(* CODESYS project OOP example Advanced Array's.project

Project tree, tasks and I/O mapping:
  Device : CODESYS Control for Raspberry Pi SL, 3S - Smart Software Solutions GmbH, version 3.5.12.30
    application Application
      libraries: Standard, * (System); VisuDialogs, * (System); SysFile, 3.5.9.0 (System); AlarmManager, 3.5.12.0 (Intern)
      task MainTask (cyclic, interval 500 ms, priority 1, watchdog 1000 ms x 1) calls Arrays
      task VISU_TASK (cyclic, interval 100 ms, priority 31) calls VisuElems.Visu_Prg
      task AlarmManagerTask (cyclic, interval 250 ms, priority 31) calls AlarmManager.Alarm_Prg
      visualisation Arrays_Visu
      program Arrays [ST]
      Alarm Configuration
        alarm class Warning (priority 10, acknowledge REP)
        AlarmStorage
        text list AlarmGroup
        alarm group AlarmGroup
            7 [Warning]: Comparison NotEqual, ExpressionToCompare 0, Expression Arrays.arEngine[7].uiAlarm - "Engine 7 Alarm"
            4 [Warning]: Comparison NotEqual, ExpressionToCompare 0, Expression Arrays.arEngine[4].uiAlarm - "Engine 4 Alarm"
            5 [Warning]: Comparison NotEqual, ExpressionToCompare 0, Expression Arrays.arEngine[5].uiAlarm - "Engine 5 Alarm"
            2 [Warning]: Comparison NotEqual, ExpressionToCompare 0, Expression Arrays.arEngine[2].uiAlarm - "Engine 2 Alarm"
            3 [Warning]: Comparison NotEqual, ExpressionToCompare 0, Expression Arrays.arEngine[3].uiAlarm - "Engine 3 Alarm"
            0 [Warning]: Comparison NotEqual, ExpressionToCompare 0, Expression Arrays.arEngine[0].uiAlarm - "Engine 0 Alarm"
            1 [Warning]: Comparison NotEqual, ExpressionToCompare 0, Expression Arrays.arEngine[1].uiAlarm - "Engine 1 Alarm"
            6 [Warning]: Comparison NotEqual, ExpressionToCompare 0, Expression Arrays.arEngine[6].uiAlarm - "Engine 6 Alarm"
    SoftMotion General Axis Pool
    I²C
    SPI
    GPIOs_A_B : GPIOs B+/Pi2, 3S - Smart Software Solutions GmbH, version 3.5.11.0
        unmapped channels: digital inputs (GPIO0..GPIO31), digital outputs (GPIO0..GPIO31)
    Onewire
    Camera device
      <Empty>
  libraries: VisuSymbols, 3.5.10.0 (System)
  Array's/
    Source/
      function block FB_Engine [ST]: Start, Stop, MaxVelocity, Temperature, Velocity
      function block FB_NewEngine [ST]: Gear, Start
      function block FB_FinalEngine [ST]: ResetAlarm, RaiseAlarm, fb_Init, Alarms
      interface ITF_AlarmSource: ResetAlarm, Alarms
      interface ITF_RaiseAlarm: RaiseAlarm
      visualisation Engine_Visu
    Handler/
      interface ITF_AlarmHandler: RegisterAlarm, ResetAllAlarms
      function block FB_AlarmHandler [ST]: RegisterAlarm, ResetAllAlarms, Registered
      interface ITF_NewAlarmHandler: RegisterAlarm, ResetAllAlarms
      function block FB_NewAlarmHandler [ST]: RegisterAlarm, ResetAllAlarms, Registered
      visualisation Handler_Visu
  text list GlobalTextList
*)

// Device/Application/Arrays
PROGRAM Arrays
VAR
	AlarmHandler : FB_NewAlarmHandler(); // The alarmhandler, which monitors all Engine's alarms
	arEngine  : ARRAY [0..10] OF FB_FinalEngine( ADR(AlarmHandler) );	// = FB_Init constructor, each engine registers itself with the alarmhandler (see method register alarm)
	
	iRegisteredAmmount : INT;
	iCnt : INT :=0;
	rVelocity : REAL := 100; //kmph
   	iGear : INT  := 5;
	xInit : BOOL := TRUE;
	xReset : BOOL := FALSE;
	xSetAlarms : BOOL := FALSE;
END_VAR

IF xInit THEN // start all engine's
	FOR iCnt := 0 TO 7 (*GVL.CUSTOM_LENGTH*) BY 1 DO
		// start engines
		arEngine[iCnt].Start(rVelocity,iGear);       //Usage of methods/properties and THIS^, see comment in method Start
	END_FOR
	xInit := FALSE;
END_IF

IF xSetAlarms THEN
	FOR iCnt := 0 TO 7 (*GVL.CUSTOM_LENGTH*) BY 1 DO
		// alarms
		arEngine[iCnt].RaiseAlarm();				// raise alarm(s)
	END_FOR
	xSetAlarms := FALSE;
END_IF

IF xReset THEN
	AlarmHandler.ResetAllAlarms();
	xReset := FALSE;
END_IF

iRegisteredAmmount := AlarmHandler.Registered;	// every registry is an alarm

END_PROGRAM

// Array's/Handler/FB_NewAlarmHandler
FUNCTION_BLOCK FB_NewAlarmHandler IMPLEMENTS ITF_AlarmHandler
VAR
	_DeviceList : ARRAY [0..7 (*GVL.CUSTOM_LENGTH*)] OF ITF_AlarmSource;
	_DeviceAmmount : INT := 0;
END_VAR

METHOD RegisterAlarm
VAR_INPUT
	DeviceWithAlarm	: ITF_AlarmSource;
END_VAR
VAR
	uiLoopIndex : INT;
END_VAR
FOR uiLoopIndex := 0 TO THIS^._DeviceAmmount - 1 DO
	IF _DeviceList[ uiLoopIndex ] = DeviceWithAlarm THEN
		RETURN;		//  Double entry => exit
	END_IF
END_FOR

// if we did not exit, it's not a double entry..
THIS^._DeviceList[ THIS^._DeviceAmmount ] := DeviceWithAlarm;
THIS^._DeviceAmmount := THIS^._DeviceAmmount + 1;
END_METHOD

METHOD ResetAllAlarms
VAR
	uiLoopIndex    : INT := 0;
END_VAR
//Resets all the alarms on each motor
FOR uiLoopIndex := 0 TO THIS^._DeviceAmmount - 1 DO
	IF _DeviceList[ uiLoopIndex ].Alarms <> 0 THEN
		_DeviceList[ uiLoopIndex ].ResetAlarm();	// pointer to all subscripted fb's Reset Methods
	END_IF
END_FOR
THIS^._DeviceAmmount := 0;
END_METHOD

// function block gekoppelde property (niet via een interface)
PROPERTY Registered : INT
GET
Registered := _DeviceAmmount;
END_GET
END_PROPERTY

END_FUNCTION_BLOCK

// Array's/Handler/ITF_AlarmHandler
INTERFACE ITF_AlarmHandler

METHOD RegisterAlarm
VAR_INPUT
	deviceWithAlarm:   ITF_AlarmSource;
END_VAR
END_METHOD

METHOD ResetAllAlarms
VAR_INPUT
END_VAR
END_METHOD

END_INTERFACE

// Array's/Source/ITF_AlarmSource
INTERFACE ITF_AlarmSource

METHOD ResetAlarm
VAR_INPUT
END_VAR
END_METHOD

//return the alarm ammount
PROPERTY Alarms : INT
GET
END_GET
END_PROPERTY

END_INTERFACE

// Array's/Source/FB_FinalEngine
FUNCTION_BLOCK FINAL FB_FinalEngine EXTENDS FB_NewEngine IMPLEMENTS ITF_AlarmSource, ITF_RaiseAlarm
VAR
   ptrAlarmHandler: POINTER TO FB_AlarmHandler;
	uiAlarm : INT := 0;	// <>0 = alarm, ideally each implemented seperate alarm raises the alarmcounter via method RaiseAlarm
END_VAR

SUPER^();

METHOD ResetAlarm
//reset the alarm (lower semaphore)
uiAlarm := uiAlarm - 1;
END_METHOD

//Alarm!
METHOD RaiseAlarm
uiAlarm := uiAlarm + 1;									// uh ohh! raise the counter, which works like a semaphore
THIS^.ptrAlarmHandler^.RegisterAlarm( THIS^ );	//register myself at handler, because we got troubles
END_METHOD

METHOD fb_Init : BOOL
VAR_INPUT
	bInitRetains : BOOL; // TRUE: the retain variables are initialized (reset warm / reset cold)
	bInCopyCode : BOOL;  // TRUE the instance will be copied to the copy-code afterward (online change)
	AlarmHandler: POINTER TO FB_AlarmHandler;		
END_VAR
THIS^.ptrAlarmHandler := AlarmHandler;		// store the handler address
END_METHOD

//return the alarm ammount
PROPERTY Alarms : INT
GET
Alarms := THIS^.uiAlarm;
END_GET
END_PROPERTY

END_FUNCTION_BLOCK

// Array's/Source/FB_NewEngine
FUNCTION_BLOCK FB_NewEngine EXTENDS FB_Engine

// HAS GOT 2 NEW Features;
// 1) START has been redefined and 
// 2) A new Gear accessor has been added
//
// these methods are fixed to the class
SUPER^();

// new property to get / set the gear after start
PROPERTY Gear : int
SET
THIS^._iGear := Gear;
END_SET
GET
Gear := THIS^._iGear;
END_GET
END_PROPERTY

METHOD Start : BOOL;
VAR_INPUT
   rVelocity : REAL;
   iGear     : INT;
END_VAR
VAR
	fVelocity: INT;
END_VAR
// Overwriting an existing method (OVERRIDE)

// new: setting gear via property Gear setter
SUPER^.Start(iGear, TO_INT(rVelocity)); // calls Start() of FB_Engine, see below for explanation
Gear := iGear;


// SUPER^. POINTER
//In the above example, we created a new Start() METHOD in FB_NewEngine 
//and copied the existing code from FB_Engine into the new method. 
//This is not always possible, and it also runs counter to the principle of reuse!
//
//Consequently, every function block which is derived from another function block has access to a pointer called SUPER. 
//This can be used to access elements (methods, properties, local variables, etc.) from the parent function block.
//
//
//SUPER^.Start(nGear, fVelocity); // calls Start() of FB_Engine
//Gear := nGear;
//
//Instead of copying code from the parent function block to the new method, 
//the SUPER pointer can be used to call the method from the FB_Engine function block. 
//This does away with the need to copy the code. 
//So, SUPER calls the Father of a method
END_METHOD

END_FUNCTION_BLOCK

// Array's/Source/FB_Engine
// Class FB_Engine
FUNCTION_BLOCK FB_Engine
VAR
   _xStarted : BOOL;
   _rVelocity : REAL;
   _rMaxVelocity : REAL;
   _iGear : INT;
   _rTemperature : REAL;
END_VAR

//The THIS pointer is available to all function blocks and points to the current function block instance. 
//It is required whenever a method contains a local variable which obscures a variable in the function block.
//
//An assignment statement within the method sets the value of the local variable. 
//If we want the method to set the value of the local variable in the function block, we need to use the THIS pointer to access it.
METHOD Start : Bool;
VAR_INPUT
   rVelocity : REAL;
   iGear     : INT;
END_VAR
THIS^._xStarted  := TRUE;
Start            := TRUE;
THIS^._iGear     := iGear;
THIS^._rVelocity := MIN( ABS(THIS^._rMaxVelocity), rVelocity );

CASE TO_INT( THIS^._rVelocity ) OF // implicit typecasting(TO_INT), use REAL_TO_INT for explicit typecasting
   0..100 :
      THIS^._rTemperature := 50;
   101..1000:
      THIS^._rTemperature := 90;
   1001..10000:
      THIS^._rTemperature := 100;
   10001..32767:
      THIS^._rTemperature := 150;
END_CASE
END_METHOD

METHOD Stop : BOOL
VAR_INPUT
END_VAR
THIS^._xStarted := FALSE;
Stop            := TRUE;
END_METHOD

PROPERTY MaxVelocity : REAL
SET
THIS^._rMaxVelocity := MaxVelocity;
END_SET
GET
MaxVelocity := THIS^._rMaxVelocity;
END_GET
END_PROPERTY

PROPERTY Temperature : REAL
GET
Temperature := THIS^._rTemperature;
END_GET
END_PROPERTY

PROPERTY Velocity : real
GET
Velocity := THIS^._rVelocity;
END_GET
END_PROPERTY

END_FUNCTION_BLOCK

// Array's/Source/ITF_RaiseAlarm
INTERFACE ITF_RaiseAlarm

METHOD RaiseAlarm
END_METHOD

END_INTERFACE

// Array's/Handler/FB_AlarmHandler
FUNCTION_BLOCK FB_AlarmHandler IMPLEMENTS ITF_AlarmHandler
VAR
	_DeviceList : ARRAY [0..99] OF ITF_AlarmSource;
	_DeviceAmmount : INT := 0;
END_VAR

METHOD RegisterAlarm
VAR_INPUT
	DeviceWithAlarm	: ITF_AlarmSource;
END_VAR
VAR
	uiLoopIndex : INT;
END_VAR
FOR uiLoopIndex := 0 TO THIS^._DeviceAmmount - 1 DO
	IF _DeviceList[ uiLoopIndex ] = DeviceWithAlarm THEN
		RETURN;		//  Double entry => exit
	END_IF
END_FOR

// if we did not exit, it's not a double entry..
THIS^._DeviceList[ THIS^._DeviceAmmount ] := DeviceWithAlarm;
THIS^._DeviceAmmount := THIS^._DeviceAmmount + 1;
END_METHOD

METHOD ResetAllAlarms
VAR
	uiLoopIndex    : INT := 0;
END_VAR
//Resets all the alarms on each motor
FOR uiLoopIndex := 0 TO THIS^._DeviceAmmount - 1 DO
	IF _DeviceList[ uiLoopIndex ].Alarms <> 0 THEN
		_DeviceList[ uiLoopIndex ].ResetAlarm();	// pointer to all subscripted fb's Reset Methods
	END_IF
END_FOR
THIS^._DeviceAmmount := 0;
END_METHOD

// function block gekoppelde property (niet via een interface)
PROPERTY Registered : INT
GET
Registered := _DeviceAmmount;
END_GET
END_PROPERTY

END_FUNCTION_BLOCK

// Array's/Handler/ITF_NewAlarmHandler
INTERFACE ITF_NewAlarmHandler

METHOD RegisterAlarm
VAR_INPUT
	deviceWithAlarm:   ITF_AlarmSource;
END_VAR
END_METHOD

METHOD ResetAllAlarms
VAR_INPUT
END_VAR
END_METHOD

END_INTERFACE

// Device/Application/Arrays_Visu
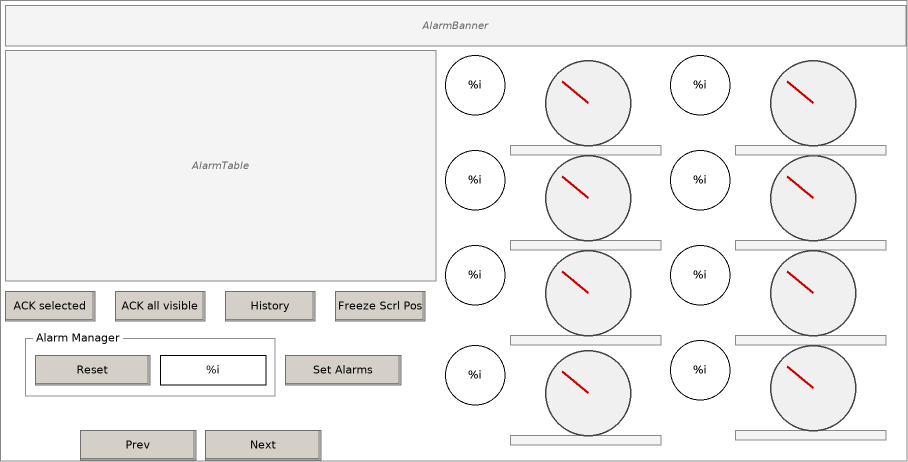
VISUALIZATION Arrays_Visu  // 908x462
VAR_IN_OUT
END_VAR
VAR
	bAckSel : BOOL;
	bAckVisible : BOOL;
	bHistory : BOOL;
	bFreezeScrlPos : BOOL;
END_VAR
    AlarmTable (5,50 431x231)
        p1521930926: __All
        p1663851261: __All
        p428520879: bAckSel
        p2607059081: bAckVisible
        p3266827225: bHistory
        p3894972949: bFreezeScrlPos
    AlarmBanner (5,5 901x41)
        p1521930926: __All
        p1663851261: __All
    Button (285,355 116x30), "Set Alarms"
        OnMouseDown: execute { Arrays.xSetAlarms := TRUE; }
    Frame (445,55 130x60)
        shows Engine_Visu(_Obj := Arrays.arEngine[0])
    Frame (445,150 141x60)
        shows Engine_Visu(_Obj := Arrays.arEngine[1])
    Frame (15,330 271x76)
        shows Handler_Visu(_Obj := Arrays.AlarmHandler)
    Frame (445,245 141x60)
        shows Engine_Visu(_Obj := Arrays.arEngine[2])
    Frame (445,345 141x60)
        shows Engine_Visu(_Obj := Arrays.arEngine[3])
    Frame (670,150 141x60)
        shows Engine_Visu(_Obj := Arrays.arEngine[5])
    Frame (670,55 141x60)
        shows Engine_Visu(_Obj := Arrays.arEngine[4])
    Frame (670,245 141x60)
        shows Engine_Visu(_Obj := Arrays.arEngine[6])
    Frame (670,340 141x61)
        shows Engine_Visu(_Obj := Arrays.arEngine[7])
    Button (5,291 90x30), "ACK selected"
        toggle bAckSel
    Button (115,291 90x30), "ACK all visible"
        toggle bAckVisible
    Button (225,291 90x30), "History"
        toggle bHistory
    Button (335,291 90x30), "Freeze Scrl Pos"
        toggle bFreezeScrlPos
    Button (205,430 116x30), "Next"
        OnMouseDown: execute { Arrays.xSetAlarms := TRUE; }
        OnMouseClick:  Type=Next
    Button (80,430 116x30), "Prev"
        OnMouseDown: execute { Arrays.xSetAlarms := TRUE; }
        OnMouseClick:  Type=Previous
END_VISUALIZATION

// Array's/Source/Engine_Visu
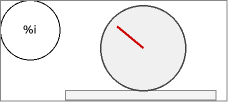
VISUALIZATION Engine_Visu  // 228x102
VAR_IN_OUT
	_Obj : FB_FinalEngine;
END_VAR
    Ellipse (0,0 60x60), "%i", text variable: _Obj._iGear, colour toggle: _Obj._xStarted
    BarDisplayImage (65,90 151x10), value: _Obj._rTemperature, style: BarDisplayImage-Gray, scale format: %.1f, scale 0..140
    Meter180 (60,5 166x86), value: _Obj._rVelocity, style: Meter-Meter180-Gray, scale format: %.1f, scale 0..220
    Ellipse (0,0 60x60), "%i", text variable: _Obj._iGear, colour toggle: _obj.uiAlarm>0
END_VISUALIZATION

// Array's/Handler/Handler_Visu
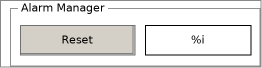
VISUALIZATION Handler_Visu  // 262x68
VAR_IN_OUT
	_Obj : FB_NewAlarmHandler;
END_VAR
    GroupBox (10,0 250x66), "Alarm Manager"
        Button (10,25 115x30), "Reset"
            OnMouseDown: execute { _Obj.ResetAllAlarms(); }
        Rectangle (135,25 106x30), "%i", text variable: _obj._DeviceAmmount, colour toggle: _obj.Registered <>0
END_VISUALIZATION

(* text list AlarmGroup (id | default)
  7 | Engine 7 Alarm
  6 | Engine 6 Alarm
  5 | Engine 5 Alarm
  4 | Engine 4 Alarm
  3 | Engine 3 Alarm
  2 | Engine 2 Alarm
  1 | Engine 1 Alarm
  0 | Engine 0 Alarm
   |  *)
